// TIA Portal V17 export
// export: Created 2022-03-12T16:05:32.6459125Z, ExportSetting WithDefaults, DisplayName Totally Integrated Automation Portal, DisplayVersion V17, DisplayName TIA Portal Openness, DisplayVersion V17, DisplayName TIA Portal Version Control Interface, DisplayVersion V17, DisplayName STEP 7 Professional, DisplayVersion V17, DisplayName STEP 7 Safety, DisplayVersion V17, DisplayName WinCC Advanced / Unified PC, DisplayVersion V17
VAR_GLOBAL   // PLC tag table "LPMLV30_Constants"
END_VAR
VAR_GLOBAL CONSTANT   // user constants
   LPMLV30_MODE_INVALID : DInt := 0;   // OMAC PackMLV30 unit mode Invalid
   LPMLV30_MODE_PRODUCTION : DInt := 1;   // OMAC PackMLV30 unit mode Production
   LPMLV30_MODE_MAINTENANCE : DInt := 2;   // OMAC PackMLV30 unit mode Maintenance
   LPMLV30_MODE_MANUAL : DInt := 3;   // OMAC PackMLV30 unit mode Manual
   LPMLV30_MODE_USER_01 : DInt := 4;   // OMAC PackMLV30 user-defined unit mode 01
   LPMLV30_MODE_USER_02 : DInt := 5;   // OMAC PackMLV30 user-defined unit mode 02
   LPMLV30_MODE_USER_03 : DInt := 6;   // OMAC PackMLV30 user-defined unit mode 03
   LPMLV30_MODE_USER_04 : DInt := 7;   // OMAC PackMLV30 user-defined unit mode 04
   LPMLV30_MODE_USER_05 : DInt := 8;   // OMAC PackMLV30 user-defined unit mode 05
   LPMLV30_MODE_USER_06 : DInt := 9;   // OMAC PackMLV30 user-defined unit mode 06
   LPMLV30_MODE_USER_07 : DInt := 10;   // OMAC PackMLV30 user-defined unit mode 07
   LPMLV30_MODE_USER_08 : DInt := 11;   // OMAC PackMLV30 user-defined unit mode 08
   LPMLV30_MODE_USER_09 : DInt := 12;   // OMAC PackMLV30 user-defined unit mode 09
   LPMLV30_MODE_USER_10 : DInt := 13;   // OMAC PackMLV30 user-defined unit mode 10
   LPMLV30_MODE_USER_11 : DInt := 14;   // OMAC PackMLV30 user-defined unit mode 11
   LPMLV30_MODE_USER_12 : DInt := 15;   // OMAC PackMLV30 user-defined unit mode 12
   LPMLV30_MODE_USER_13 : DInt := 16;   // OMAC PackMLV30 user-defined unit mode 13
   LPMLV30_MODE_USER_14 : DInt := 17;   // OMAC PackMLV30 user-defined unit mode 14
   LPMLV30_MODE_USER_15 : DInt := 18;   // OMAC PackMLV30 user-defined unit mode 15
   LPMLV30_MODE_USER_16 : DInt := 19;   // OMAC PackMLV30 user-defined unit mode 16
   LPMLV30_MODE_USER_17 : DInt := 20;   // OMAC PackMLV30 user-defined unit mode 17
   LPMLV30_MODE_USER_18 : DInt := 21;   // OMAC PackMLV30 user-defined unit mode 18
   LPMLV30_MODE_USER_19 : DInt := 22;   // OMAC PackMLV30 user-defined unit mode 19
   LPMLV30_MODE_USER_20 : DInt := 23;   // OMAC PackMLV30 user-defined unit mode 20
   LPMLV30_MODE_USER_21 : DInt := 24;   // OMAC PackMLV30 user-defined unit mode 21
   LPMLV30_MODE_USER_22 : DInt := 25;   // OMAC PackMLV30 user-defined unit mode 22
   LPMLV30_MODE_USER_23 : DInt := 26;   // OMAC PackMLV30 user-defined unit mode 23
   LPMLV30_MODE_USER_24 : DInt := 27;   // OMAC PackMLV30 user-defined unit mode 24
   LPMLV30_MODE_USER_25 : DInt := 28;   // OMAC PackMLV30 user-defined unit mode 25
   LPMLV30_MODE_USER_26 : DInt := 29;   // OMAC PackMLV30 user-defined unit mode 26
   LPMLV30_MODE_USER_27 : DInt := 30;   // OMAC PackMLV30 user-defined unit mode 27
   LPMLV30_MODE_USER_28 : DInt := 31;   // OMAC PackMLV30 user-defined unit mode 28
   LPMLV30_STATE_UNDEFINED : DInt := 0;   // OMAC PackMLV30 state Undefined
   LPMLV30_STATE_CLEARING : DInt := 1;   // OMAC PackMLV30 state Clearing
   LPMLV30_STATE_STOPPED : DInt := 2;   // OMAC PackMLV30 state Stopped
   LPMLV30_STATE_STARTING : DInt := 3;   // OMAC PackMLV30 state Starting
   LPMLV30_STATE_IDLE : DInt := 4;   // OMAC PackMLV30 state Idle
   LPMLV30_STATE_SUSPENDED : DInt := 5;   // OMAC PackMLV30 state Suspended
   LPMLV30_STATE_EXECUTE : DInt := 6;   // OMAC PackMLV30 state Execute
   LPMLV30_STATE_STOPPING : DInt := 7;   // OMAC PackMLV30 state Stopping
   LPMLV30_STATE_ABORTING : DInt := 8;   // OMAC PackMLV30 state Aborting
   LPMLV30_STATE_ABORTED : DInt := 9;   // OMAC PackMLV30 state Aborted
   LPMLV30_STATE_HOLDING : DInt := 10;   // OMAC PackMLV30 state Holding
   LPMLV30_STATE_HELD : DInt := 11;   // OMAC PackMLV30 state Held
   LPMLV30_STATE_UNHOLDING : DInt := 12;   // OMAC PackMLV30 state Unholding
   LPMLV30_STATE_SUSPENDING : DInt := 13;   // OMAC PackMLV30 state Suspending
   LPMLV30_STATE_UNSUSPENDING : DInt := 14;   // OMAC PackMLV30 state Unsuspending
   LPMLV30_STATE_RESETTING : DInt := 15;   // OMAC PackMLV30 state Resetting
   LPMLV30_STATE_COMPLETING : DInt := 16;   // OMAC PackMLV30 state Completing
   LPMLV30_STATE_COMPLETE : DInt := 17;   // OMAC PackMLV30 state Complete
   LPMLV30_CMD_UNDEFINED : DInt := 0;   // OMAC PackMLV30 control command Undefined
   LPMLV30_CMD_RESET : DInt := 1;   // OMAC PackMLV30 control command Reset
   LPMLV30_CMD_START : DInt := 2;   // OMAC PackMLV30 control command Start
   LPMLV30_CMD_STOP : DInt := 3;   // OMAC PackMLV30 control command Stop
   LPMLV30_CMD_HOLD : DInt := 4;   // OMAC PackMLV30 control command Hold
   LPMLV30_CMD_UNHOLD : DInt := 5;   // OMAC PackMLV30 control command Unhold
   LPMLV30_CMD_SUSPEND : DInt := 6;   // OMAC PackMLV30 control command Suspend
   LPMLV30_CMD_UNSUSPEND : DInt := 7;   // OMAC PackMLV30 control command Unsuspend
   LPMLV30_CMD_ABORT : DInt := 8;   // OMAC PackMLV30 control command Abort
   LPMLV30_CMD_CLEAR : DInt := 9;   // OMAC PackMLV30 control command Clear
   LPMLV30_CMD_COMPLETE : DInt := 10;   // OMAC PackMLV30 control command Complete
   LPMLV30_LANGUAGE_1 : Int := 0;   // Texts in 1st language (default English)
   LPMLV30_LANGUAGE_2 : Int := 1;   // Texts in 2nd language (default German)
   LPMLV30_DIAG_BUFFER_UPPER_LIM : Int := 15;   // Diagnostics buffer array upper boundary (0-based)
   LPMLV30_LANGUAGES_UPPER_LIM : Int := 2;   // (Number of languages - 1) -> Array[0..LPMLV30_LANGUAGES_UPPER_LIM]
   LPMLV30_MODES_UPPER_LIM : Int := 4;   // (Number of unit modes - 1) -> Array[0..LPMLV30_MODES_UPPER_LIM]
   LPMLV30_STATES_UPPER_LIM : Int := 17;   // (Number of states - 1) -> Array[0..LPMLV30_STATES_UPPER_LIM] (SHOULD ALWAYS BE 17!)
   LPMLV30_MAX_MODES_UPPER_LIM : Int := 31;   // (Maximum number of unit modes - 1) -> Array[0..LPMLV30_MAX_MODES_UPPER_LIM]
END_VAR
